(* IEC 61131-3 sources: teller/JD_Teller_LC2_V11/Class/Pulser, 1 file *)

(* ---- Pulser.st ---- *)
(*!
<Class
	Name               = "Pulser"
	Revision           = "1.1"
	RealtimeTask       = "false"
	CyclicTask         = "true"
	BackgroundTask     = "false"
	Sigmatek           = "false"
	OSInterface        = "false"
	HighPriority       = "false"
	Automatic          = "false"
	UpdateMode         = "Prescan"
	SharedCommandTable = "true"
	Objectsize         = "(284,120)">
	<Channels>
		<Server Name="ClassSvr" Visualized="false" Initialize="false" WriteProtected="true" Retentive="false"/>
		<Client Name="ResetIn" Required="true" Internal="false"/>
		<Client Name="ResetOut" Required="true" Internal="false"/>
	</Channels>
	<RevDoku>
		<Owner Company="JD" Author="Johannes"/>
		<Dokumentation Revision="1.1" Date="2013-09-25" Author="Johannes" Company="JD" Description="Code aangepast, zelfde functie"/>
		<Dokumentation Revision="1.0" Date="2011-09-01" Author="Johannes" Company="JD" Description="Reset duur op 4 seconden"/>
	</RevDoku>
</Class>
*)
Pulser : CLASS
  //Servers:
	ClassSvr 	: SvrChCmd_DINT;
  //Clients:
	ResetIn 	: CltCh_DINT;
	ResetOut 	: CltCh_DINT;
  //Variables:
		Timer 	: UDINT;
		CasePulser 	: DINT;
		ResetOutOld 	: DINT;
  //Functions:

	FUNCTION VIRTUAL GLOBAL Init;

	FUNCTION VIRTUAL GLOBAL CyWork
		VAR_INPUT
			EAX 	: UDINT;
		END_VAR
		VAR_OUTPUT
			state (EAX) 	: UDINT;
		END_VAR;
  //Tables:
	FUNCTION @STD
		VAR_OUTPUT
			ret_code	: CONFSTATES;
		END_VAR;
	FUNCTION GLOBAL TAB @CT_;
END_CLASS;

FUNCTION VIRTUAL GLOBAL Pulser::Init

if _FirstScan then

end_if;

END_FUNCTION

FUNCTION VIRTUAL GLOBAL Pulser::CyWork
	VAR_INPUT
		EAX 	: UDINT;
	END_VAR
	VAR_OUTPUT
		state (EAX) 	: UDINT;
	END_VAR

  ResetIn := ResetIn.Read();

  if    ResetIn = 1 then

        case CasePulser of

        0:

            Timer := ops.tAbsolute;
            ResetOut := 0;
            CasePulser := 1;

        1:
            if    ops.tAbsolute - timer < 2000 then
                  if    ResetOut = 1 then
                        ResetOut := 0;
                  else
                        ResetOut := 1;
                  end_if;
            else
                  CasePulser := 2;

            end_if;

        2:
            //doe niets
            ResetOut := 0;
        end_case;

  else
        CasePulser := 0;
        ResetOut := 0;
  end_if;

  if    ResetOut <> ResetOutOld   then
        ResetOutOld := ResetOut;
        ResetOut.Write(ResetOut);
  end_if;

	state := READY;

END_FUNCTION
